// TIA Portal project "Pneumatic" (V15)

(* hardware
DEVICE "S7-1200 station_1"  S7-1200 Station
   slot 0: "Rack_0"  S7-1200 Rack  Rack  V1.0
   slot 1: "PLC_1"  CPU 1214C DC/DC/DC  6ES7 214-1AG40-0XB0  V4.2
*)

// ===== PLC "PLC_1"  CPU 1214C DC/DC/DC =====

VAR_GLOBAL   // PLC tag table "Default tag table"
   "START" AT %I0.1 : Bool;
   "STOP" AT %I0.0 : Bool;
   "R1" AT %Q0.0 : Bool;
   "R2" AT %Q0.1 : Bool;
   "R3" AT %Q0.2 : Bool;
   "H2" AT %Q0.3 : Bool;
   "H3" AT %Q0.4 : Bool;
   "Tag_8" AT %I0.3 : Bool;
   "OLR" AT %I0.2 : Bool;
   "H1" AT %Q0.5 : Bool;
END_VAR

// folder: System blocks/Program resources

DATA_BLOCK "T0"   // DB1
{ S7_Optimized_Access := 'TRUE' }
AUTHOR : Simatic
FAMILY : IEC
NAME : IEC_TMR
VERSION : 1.0
// stored: InstanceOfName IEC_TIMER
"IEC_TIMER"
BEGIN
END_DATA_BLOCK

// folder: (top level)

ORGANIZATION_BLOCK "Main"   // OB1, LAD, ProgramCycle
TITLE = "Main Program Sweep (Cycle)"
{ S7_Optimized_Access := 'TRUE' }
VERSION : 0.1
   VAR_INPUT
      Initial_Call : Bool;   // Initial call of this OB
      Remanence : Bool;   // =True, if remanent data are available
   END_VAR
BEGIN

REGION Network 1
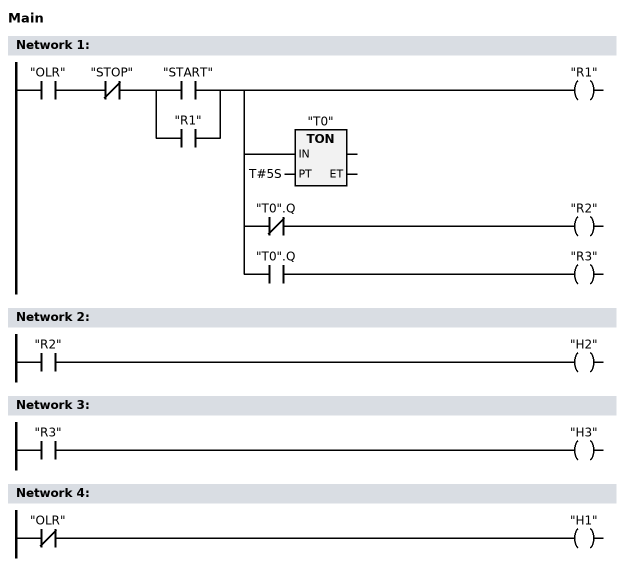
   "R1" := "OLR" AND NOT "STOP" AND ("START" OR "R1");
   "T0".TON(IN := "R1", PT := T#5S);
   "R2" := "R1" AND NOT "T0".Q;
   "R3" := "R1" AND "T0".Q;
END_REGION

REGION Network 2
   RUNG wire#powerrail
      Contact( "R2" )
      Coil( "H2" )
   END_RUNG
   // the same network as SCL:
   "H2" := "R2";
END_REGION

REGION Network 3
   RUNG wire#powerrail
      Contact( "R3" )
      Coil( "H3" )
   END_RUNG
   // the same network as SCL:
   "H3" := "R3";
END_REGION

REGION Network 4
   RUNG wire#powerrail
      I_Contact( "OLR" )
      Coil( "H1" )
   END_RUNG
   // the same network as SCL:
   "H1" := NOT "OLR";
END_REGION
END_ORGANIZATION_BLOCK